(* IEC 61131-3 sources: Industry-PLC-LLM/data/PLCBEAD_repo/PLCBEAD_PLCEmbed-main/PLC-BEAD/Source/GEB/SWAP_BYTE2, 1 file *)

(* ---- SWAP_BYTE2.ST ---- *)
FUNCTION SWAP_BYTE2:DWORD

	VAR_INPUT
		INPUT :	DWORD;
	END_VAR

	Swap_Byte2 := (ROR(INPUT,8) AND DWORD#16#FF00FF00) OR (ROL(INPUT,8) AND DWORD#16#00FF00FF);

END_FUNCTION

PROGRAM program0

	VAR
		IN :	DWORD;
		CEIL5_OUT : DWORD;
	END_VAR

	CEIL5_OUT := SWAP_BYTE2(IN);

END_PROGRAM
